PROGRAM prgLab14B
VAR
	r1:REAL:=10;
	r2:REAL:=1;
	r3:REAL;
	b1 AT %I*:BOOL;
END_VAR

IF b1 THEN
	r2:=0;
END_IF

r3:=r1/r2;

END_PROGRAM

(* stored: Version 1.1.0.1, ProductVersion 3.1.4024.11
   POU prgLab14B: Id {54dd10cf-42c1-4320-ba74-0149af57acea}, SpecialFunc None *)
